FUNCTION_BLOCK imageNormalizationFunction

VAR_IN_OUT
	imageMatrix: ARRAY[1..constants.IMG_WIDTH, 1..constants.IMG_HEIGHT] OF REAL;
END_VAR

VAR_INPUT
	start: BOOL;
END_VAR

VAR_OUTPUT
	error: BOOL;
	finished: BOOL := FALSE;
END_VAR

VAR
	x: UDINT;
	y: UDINT;
	normalizationFactor: REAL := 255.0;
END_VAR

	
IF (start) AND (NOT finished) THEN
	
	FOR x := 1 TO constants.IMG_WIDTH DO
		FOR y := 1 TO constants.IMG_HEIGHT DO
			
			imageMatrix[x, y] := imageMatrix[x, y] / normalizationfactor;
			
		END_FOR
	END_FOR
	
	finished := TRUE;
	 
END_IF

END_FUNCTION_BLOCK

(* stored: Version 1.1.0.1
   POU imageNormalizationFunction: Id {4fe8d203-47f6-4c64-9131-0c60395d5c06}, SpecialFunc None *)
